# EPICS substitutions: iocbio4/iocBoot/digital_O.substitutions
#file stdApp/Db/digital_O.db
file "$(TOP)/18IDdApp/Db/digital_O.db"
{
	pattern { id, C, S }

        { 18ID, 0,  0 }
        { 18ID, 0,  1 }
        { 18ID, 0,  2 }
        { 18ID, 0,  3 }
        { 18ID, 0,  4 }
        { 18ID, 0,  5 }
        { 18ID, 0,  6 }
        { 18ID, 0,  7 }
        { 18ID, 0,  8 }
        { 18ID, 0,  9 }
        { 18ID, 0, 10 }
        { 18ID, 0, 11 }
        { 18ID, 0, 12 }
        { 18ID, 0, 13 }
        { 18ID, 0, 14 }
        { 18ID, 0, 15 }
}
